// TIA Portal V19 export
DATA_BLOCK "A0201_Profilatrice_RegolazioneFormato"   // DB47
// stored: InstanceOfName A0201_Profilatrice_RegolazioneFormato_FB, InstanceOfType FB
"A0201_Profilatrice_RegolazioneFormato_FB"
   // VAR_INPUT
   //    AreaInterface : "AreaInterface";
   //    ZSI : "udt_ZoneSafetyInterface";
   //    DSI : Array[1..14] of "udt_DeviceSafetyInterface";
   //    Cin : Struct
   //       LineSetup_Exe : Bool;
   //       OB30_High : Bool;
   //       Infeed_ON : Bool;
   //    END_STRUCT;
   //    DataIn : Struct
   //       PB_Passaggio02_Combo : "Ax_PB";
   //       PB_Passaggio14_Combo : "Ax_PB";
   //       PB_Passaggio17_Combo : "Ax_PB";
   //       PB_Passaggio18_Combo : "Ax_PB";
   //    END_STRUCT;
   // END_VAR
   // VAR_OUTPUT
   //    MachineInterface { ExternalAccessible := 'False'; ExternalVisible := 'False'; ExternalWritable := 'False'} : "MachineInterface";
   //    Cout : Struct
   //       OB30_High_Req : Bool;
   //       Infeed_ReqON : Bool;
   //       CtrlSafe_AX_M : Bool;
   //       SetUp_Done : Array[1..14] of Bool;
   //    END_STRUCT;
   // END_VAR
   // VAR_IN_OUT
   //    Par_Machne : Struct
   //       Passaggio02_MaxDisallineamentoAXs : Real;
   //       Passaggio14_MaxDisallineamentoAXs : Real;
   //       Passaggio17_MaxDisallineamentoAXs : Real;
   //       Passaggio18_MaxDisallineamentoAXs : Real;
   //       AxD_AutoSpeed : Real;
   //    END_STRUCT;
   //    Par_Enc : Array[1..14] of "PosFbk_RTN";
   //    Par_D : Array[1..6] of "Positioning_DOL_Machine_Par";
   //    Par_M : Array[7..14] of "Positioning_MOL_Machine_Par";
   //    Pers_D : Array[1..6] of "Positioning_DOL_Machine_Pers_Data";
   //    Pers_M : Array[7..14] of "Positioning_MOL_Machine_Pers_Data";
   // END_VAR
   // VAR
   //    i : Int;
   //    Init_Done : Bool;
   //    HMI : Struct
   //       Passaggio02_Combo_TargetPos : Real;
   //       Passaggio14_Combo_TargetPos : Real;
   //       Passaggio17_Combo_TargetPos : Real;
   //       Passaggio18_Combo_TargetPos : Real;
   //    END_STRUCT;
   //    Warning : Struct
   //       Ax_D { S7_SetPoint := 'True'} : Array[1..6] of "Positioning_DOL_Machine_Wng";
   //       Ax_M : Array[7..14] of "Positioning_MOL_Machine_Wng";
   //       Passaggio02_MaxDisallineamentoAXs { S7_SetPoint := 'True'} : Bool;
   //       Passaggio14_MaxDisallineamentoAXs { S7_SetPoint := 'True'} : Bool;
   //       Passaggio17_MaxDisallineamentoAXs { S7_SetPoint := 'True'} : Bool;
   //       Passaggio18_MaxDisallineamentoAXs { S7_SetPoint := 'True'} : Bool;
   //    END_STRUCT;
   //    Alarm : Struct
   //       Enc : Array[1..14] of "PosFbk_Encoder_Alr";
   //       Ax_D { S7_SetPoint := 'True'} : Array[1..6] of "Positioning_DOL_Machine_Alr";
   //       Ax_M { S7_SetPoint := 'True'} : Array[7..14] of "Positioning_MOL_Machine_Alr";
   //    END_STRUCT;
   //    Sts : Struct
   //       UpdateSel : Int;
   //       Passaggio02 : Struct
   //          DeltaPos_OP_MOT : LReal;
   //          AxOP_Pause_Minus : Bool;
   //          AxOP_Pause_Plus : Bool;
   //          AxMOT_Pause_Minus : Bool;
   //          AxMOT_Pause_Plus : Bool;
   //       END_STRUCT;
   //       Passaggio14 : Struct
   //          DeltaPos_OP_MOT : LReal;
   //          AxOP_Pause_Minus : Bool;
   //          AxOP_Pause_Plus : Bool;
   //          AxMOT_Pause_Minus : Bool;
   //          AxMOT_Pause_Plus : Bool;
   //       END_STRUCT;
   //       Passaggio17 : Struct
   //          DeltaPos_OP_MOT : LReal;
   //          AxOP_Pause_Minus : Bool;
   //          AxOP_Pause_Plus : Bool;
   //          AxMOT_Pause_Minus : Bool;
   //          AxMOT_Pause_Plus : Bool;
   //       END_STRUCT;
   //       Passaggio18 : Struct
   //          DeltaPos_OP_MOT : LReal;
   //          AxOP_Pause_Minus : Bool;
   //          AxOP_Pause_Plus : Bool;
   //          AxMOT_Pause_Minus : Bool;
   //          AxMOT_Pause_Plus : Bool;
   //       END_STRUCT;
   //       TargetPos : Array[1..14] of Real;
   //    END_STRUCT;
   //    Ctrl : Struct
   //       OB30_High_Req : Bool;
   //       Passaggio02_Combo_MAN : Struct
   //          Minus : Bool;
   //          Plus : Bool;
   //          MoveToPos : Bool;
   //       END_STRUCT;
   //       Passaggio14_Combo_MAN : Struct
   //          Minus : Bool;
   //          Plus : Bool;
   //          MoveToPos : Bool;
   //       END_STRUCT;
   //       Passaggio17_Combo_MAN : Struct
   //          Minus : Bool;
   //          Plus : Bool;
   //          MoveToPos : Bool;
   //       END_STRUCT;
   //       Passaggio18_Combo_MAN : Struct
   //          Minus : Bool;
   //          Plus : Bool;
   //          MoveToPos : Bool;
   //       END_STRUCT;
   //    END_STRUCT;
   //    EncITF : Array[1..14] of "PosFbk_ITF";
   //    TOF_OB30_High { S7_SetPoint := 'True'} : TOF_TIME;
   //    Enc { S7_SetPoint := 'True'} : Array[1..14] of "PosFbk_SickAFM60";
   //    AX_D { S7_SetPoint := 'True'} : Array[1..6] of "Positioning_DOL_Machine_FB";
   //    AX_M { S7_SetPoint := 'True'} : Array[7..14] of "Positioning_MOL_Machine_FB";
   //    AUX : Struct
   //       PB_Passaggio02_Combo : Struct
   //          Minus : Bool;
   //          Plus : Bool;
   //          MoveToPos : Bool;
   //       END_STRUCT;
   //       PB_Passaggio14_Combo : Struct
   //          Minus : Bool;
   //          Plus : Bool;
   //          MoveToPos : Bool;
   //       END_STRUCT;
   //       PB_Passaggio17_Combo : Struct
   //          Minus : Bool;
   //          Plus : Bool;
   //          MoveToPos : Bool;
   //       END_STRUCT;
   //       PB_Passaggio18_Combo : Struct
   //          Minus : Bool;
   //          Plus : Bool;
   //          MoveToPos : Bool;
   //       END_STRUCT;
   //    END_STRUCT;
   // END_VAR
BEGIN
END_DATA_BLOCK
